// SIMATIC S7-200 project (STEP 7-Micro/WIN), CPU 224XP CN REL 02.01

ORGANIZATION_BLOCK 程序块:OB1
TITLE=程序注释
BEGIN
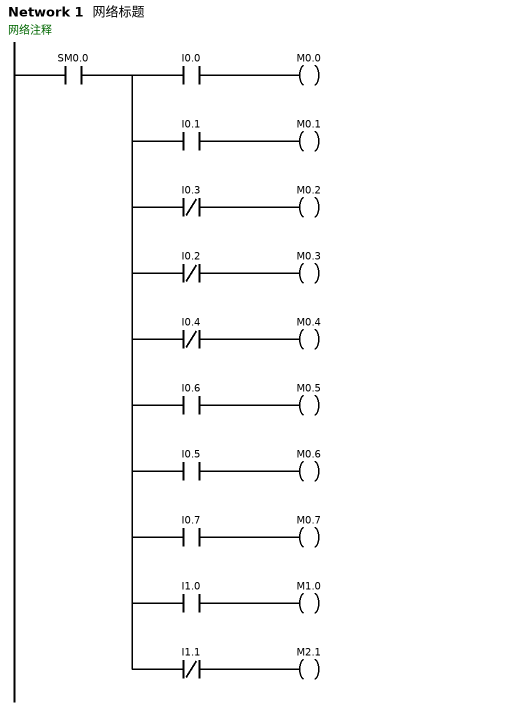
Network 1 // 网络标题
// 网络注释
LD     SM0.0
LPS
A      I0.0
=      M0.0
LRD
A      I0.1
=      M0.1
LRD
AN     I0.3
=      M0.2
LRD
AN     I0.2
=      M0.3
LRD
AN     I0.4
=      M0.4
LRD
A      I0.6
=      M0.5
LRD
A      I0.5
=      M0.6
LRD
A      I0.7
=      M0.7
LRD
A      I1.0
=      M1.0
LPP
AN     I1.1
=      M2.1
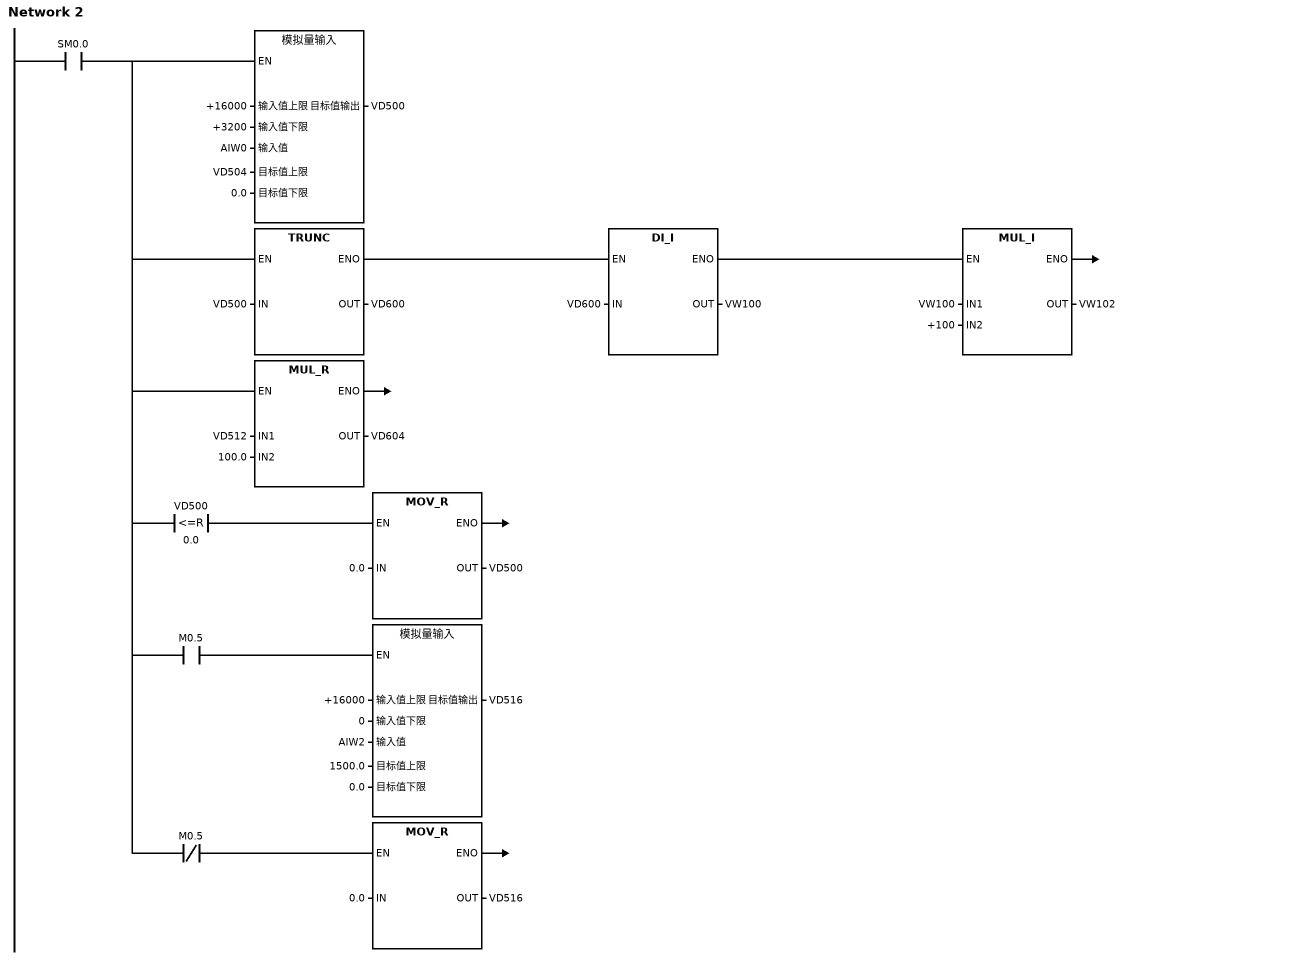
Network 2
LD     SM0.0
LPS
CALL   模拟量输入:SBR2, +16000, +3200, AIW0, VD504, 0.0, VD500
TRUNC  VD500, VD600
AENO
DTI    VD600, VW100
AENO
MOVW   VW100, VW102
*I     +100, VW102
LRD
MOVR   VD512, VD604
*R     100.0, VD604
LRD
AR<=   VD500, 0.0
MOVR   0.0, VD500
LRD
A      M0.5
CALL   模拟量输入:SBR2, +16000, 0, AIW2, 1500.0, 0.0, VD516
LPP
AN     M0.5
MOVR   0.0, VD516
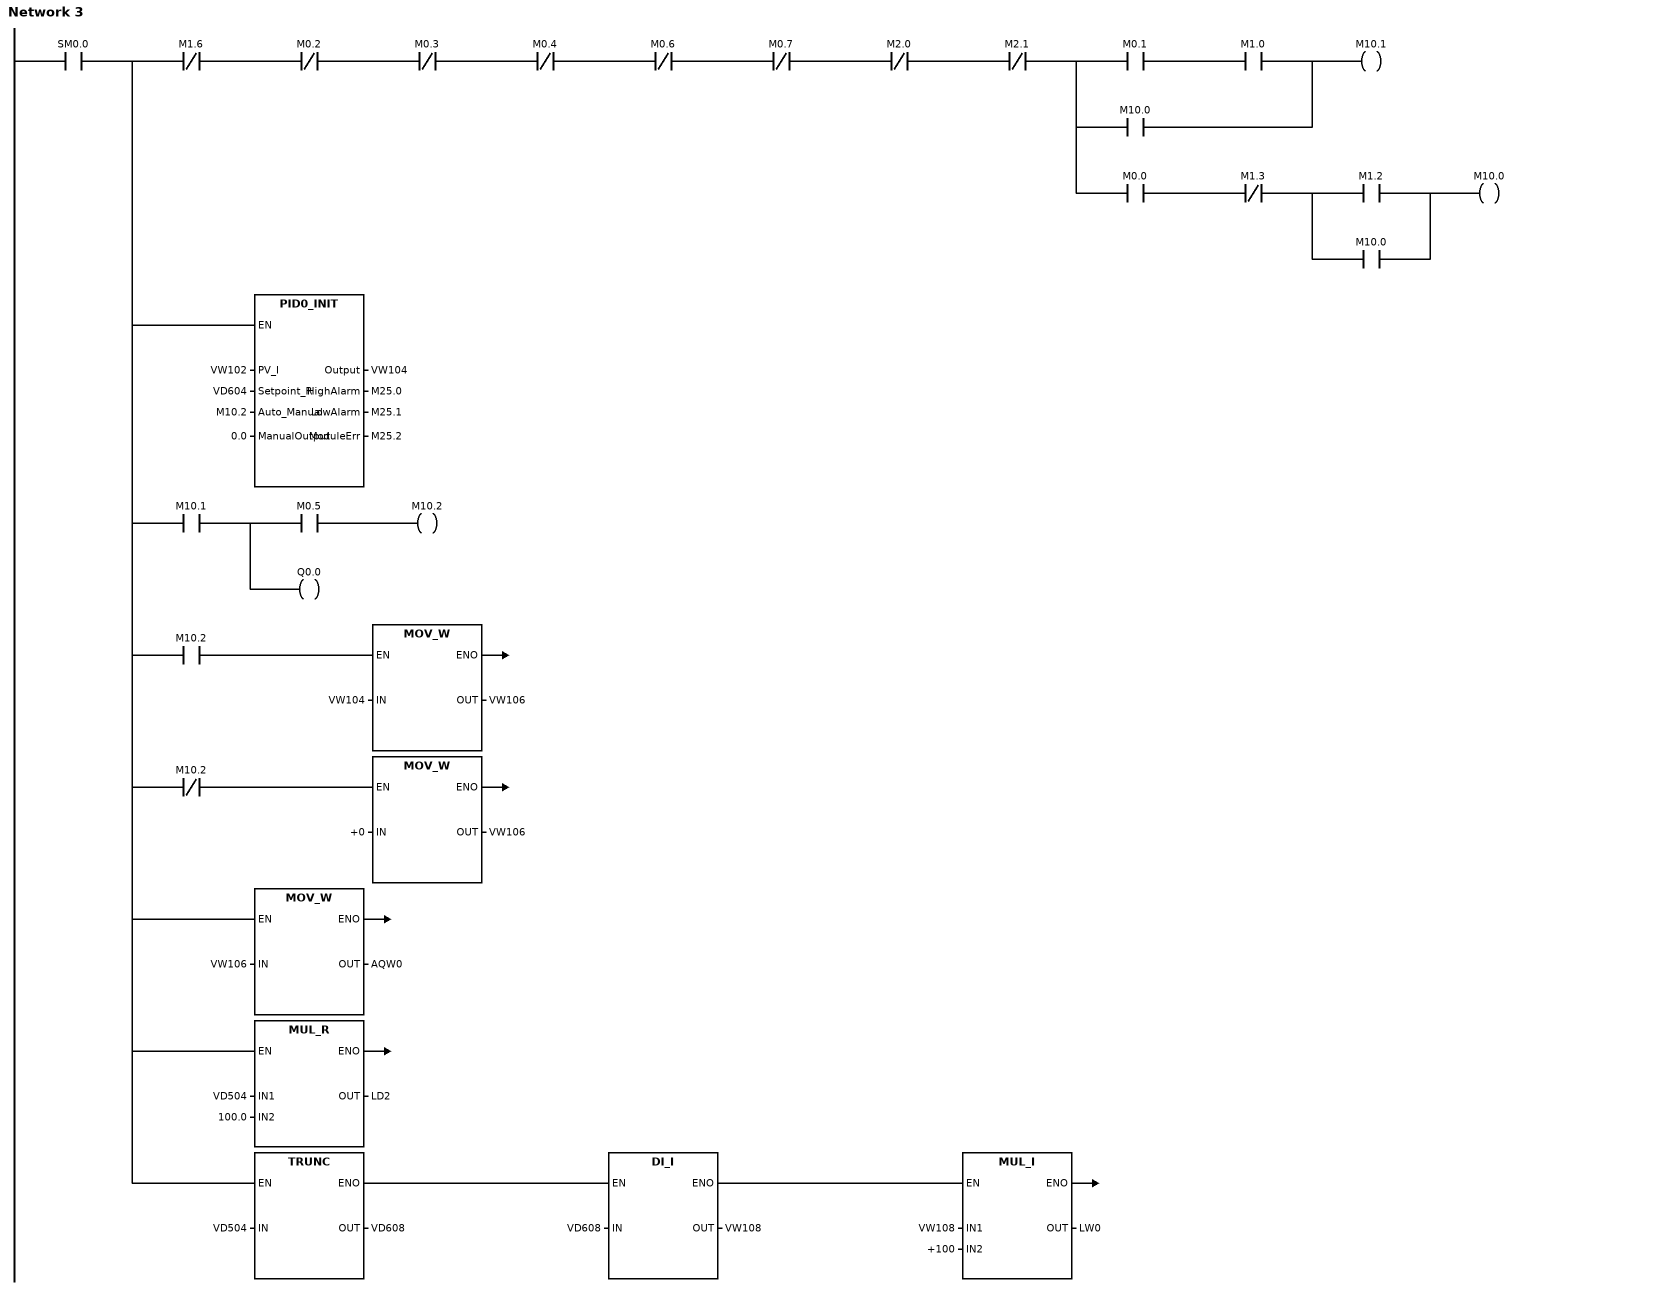
Network 3
LD     SM0.0
LPS
AN     M1.6
AN     M0.2
AN     M0.3
AN     M0.4
AN     M0.6
AN     M0.7
AN     M2.0
AN     M2.1
LPS
LD     M0.1
A      M1.0
O      M10.0
ALD
=      M10.1
LPP
A      M0.0
AN     M1.3
LD     M1.2
O      M10.0
ALD
=      M10.0
LPP
LPS
CALL   PID0_INIT:SBR4, VW102, VD604, M10.2, 0.0, VW104, M25.0, M25.1, M25.2
A      M10.1
LPS
A      M0.5
=      M10.2
LPP
=      Q0.0
LPP
LPS
A      M10.2
MOVW   VW104, VW106
LRD
AN     M10.2
MOVW   +0, VW106
LRD
MOVW   VW106, AQW0
LRD
MOVR   VD504, LD2
*R     100.0, LD2
LPP
TRUNC  VD504, VD608
AENO
DTI    VD608, VW108
AENO
MOVW   VW108, LW0
*I     +100, LW0
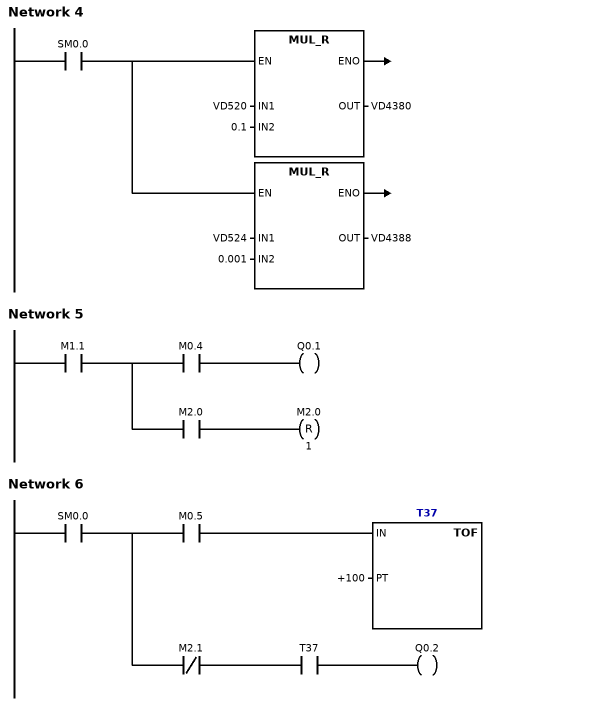
Network 4
LD     SM0.0
MOVR   VD520, VD4380
*R     0.1, VD4380
MOVR   VD524, VD4388
*R     0.001, VD4388
Network 5
LD     M1.1
LPS
A      M0.4
=      Q0.1
LPP
A      M2.0
R      M2.0, 1
Network 6
LD     SM0.0
LPS
A      M0.5
TOF    T37, +100
LPP
AN     M2.1
A      T37
=      Q0.2
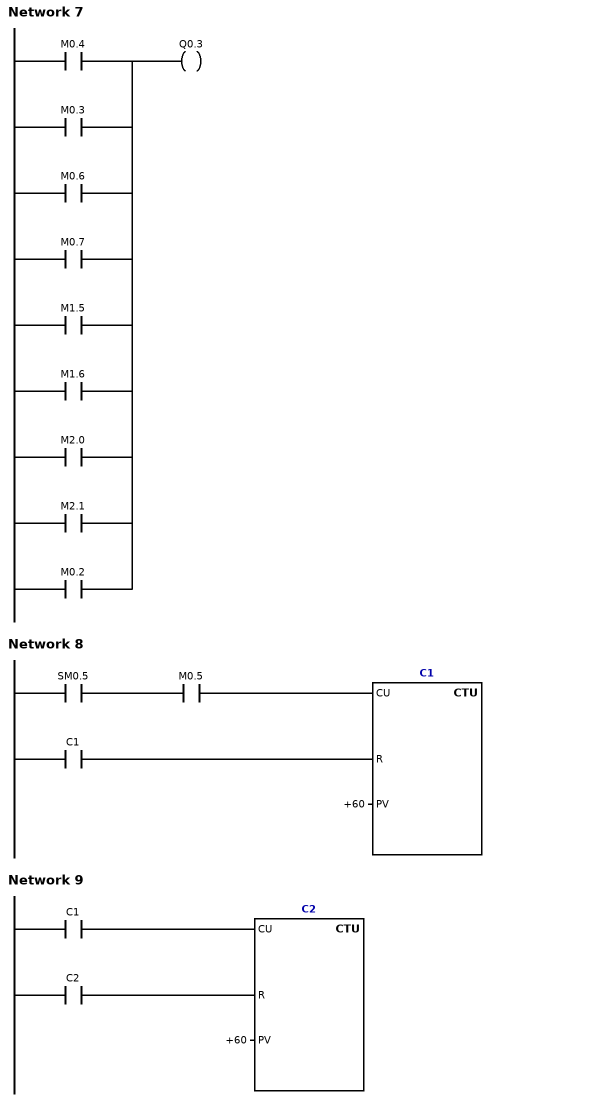
Network 7
LD     M0.4
O      M0.3
O      M0.6
O      M0.7
O      M1.5
O      M1.6
O      M2.0
O      M2.1
O      M0.2
=      Q0.3
Network 8
LD     SM0.5
A      M0.5
LD     C1
CTU    C1, +60
Network 9
LD     C1
LD     C2
CTU    C2, +60
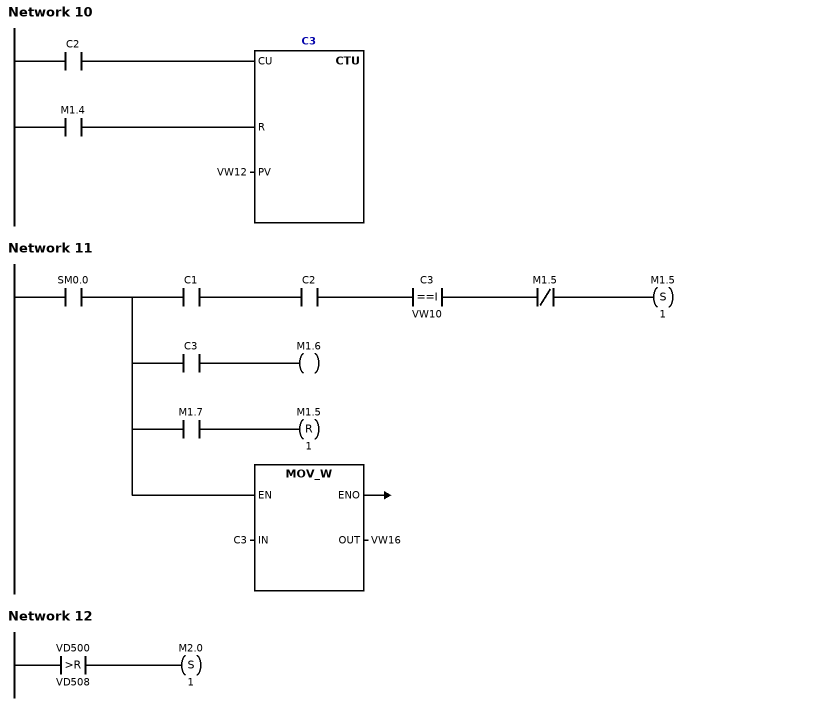
Network 10
LD     C2
LD     M1.4
CTU    C3, VW12
Network 11
LD     SM0.0
LPS
A      C1
A      C2
AW=    C3, VW10
AN     M1.5
S      M1.5, 1
LRD
A      C3
=      M1.6
LRD
A      M1.7
R      M1.5, 1
LPP
MOVW   C3, VW16
Network 12
LDR>   VD500, VD508
S      M2.0, 1
END_ORGANIZATION_BLOCK

// SBR2: protected block, not included

// SBR4: protected block, not included

// INT0: protected block, not included

// (further data pages could not be read)
